TYPE ST_CYLINDER_Status :
STRUCT

	I					: ST_CYLINDER_IN;
	Q					: ST_CYLINDER_OUT;

END_STRUCT
END_TYPE

(* stored: Version 1.1.0.1
   DUT ST_CYLINDER_Status: Id {bf1b356b-8ff7-4fb7-9eba-e3f9c25b161e} *)
